// TIA Portal V20 export
TYPE "LKinCtrl_typeMovePathDiagnostics"
   STRUCT
      errorID : Word;   // errorID of the FB
      pathDataName : String["LKINCTRL_LENGTH_OF_PATHDATA_NAME"];   // name of PathData an error occurred in
      cmdNumber : DInt;   // command number (in PathData) an error occurred in
      stateMovePath : DInt;   // state machine status FB
      statusSubFunction : Word;   // status of LKinCtrl_MC_ExecuteKinMotionCmd
      motionFBNumber : DInt;   // motion FB number (internal) an error occurred in
      motionFBStatus : DWord;   // status of motion FB (internal) an error occurred in
      kinematicsStatusWord : DWord;   // statusWord TO kinematics
      kinematicsErrorWord : DWord;   // errorWord TO kinematics
   END_STRUCT;
END_TYPE
